Universal Robots PolyScope program: align_for_step.urp

Program align_for_step (installation=default directory=/programs createdIn=5.21.3 lastSavedIn=5.21.3 robotSerialNumber=20246801938)
Calibrated DH parameters: a=[-0.000071, -0.790281, -0.600694, 0.000061, -0.000039, 0]; d=[0.236272, 604.465945, 132.116513, -736.382239, 0.159268, 0.154005]; alpha=[1.570254, -0.000567, 0.000559, 1.571709, -1.56999, 0]; deltaTheta=[0, -0.409357, 7.293326, -0.600784, -0.000001, -0.000001]
InitVariablesNode
Robot Program (runOnlyOnce=false)
  'first move block is unnecessay and bad'
  SuppressedNode
    MoveJ speed 60 deg/s, acceleration 80 deg/s^2 (useActiveTCP=true optimoveEnabled=false optiMoveSpeed=0.3 optiMoveAcceleration=0.09) feature=Base
      'belowis oldhome'
      Waypoint Waypoint_1: TCP in base x=397.354 y=356.263 z=319.809 mm, rx=2.3163 ry=2.0576 rz=0.0741 rad; joints [-198.308, -118.162, 133.452, -12.561, -11.517, -6.326] deg; TCP offset x=-9.5 y=-328 z=105.73 mm, rx=1.2092 ry=-1.2092 rz=1.2092 rad
      SuppressedNode
        Waypoint Waypoint_2: TCP in base x=102.072 y=804.129 z=-21.158 mm, rx=-1.0098 ry=-2.9661 rz=0.0347 rad; joints [-131.791, -72.228, 126.432, -52.794, -4.122, -0.058] deg
      SuppressedNode
        Waypoint Waypoint_3: TCP in base x=-481.576 y=738.776 z=-387.745 mm, rx=-0.0268 ry=3.1371 rz=-0.1325 rad; joints [-88.373, -42.244, 121.849, -79.055, 0.705, 4.289] deg
      Waypoint Waypoint_4: TCP in base x=-790.625 y=220.046 z=-730.503 mm, rx=-0.9425 ry=2.9648 rz=-0.1356 rad; joints [-49.775, -15.59, 117.776, -102.401, 4.996, 5.448] deg
      Waypoint Waypoint_5: TCP in base x=-802.158 y=237.168 z=-730.663 mm, rx=0.8868 ry=-2.4516 rz=0.2829 rad; joints [-61.24, 14.733, 101.407, -222.645, 33.575, 110.967] deg
      Waypoint Waypoint_6: TCP in base x=-687.678 y=589.975 z=-233.622 mm, rx=-0.3444 ry=-1.0001 rz=-2.0808 rad; joints [-61.24, 14.733, 101.407, -222.645, 33.575, -30.853] deg
      SuppressedNode
        Waypoint goalpt: TCP in base x=-796.965 y=229.005 z=-75.004 mm, rx=0 ry=0 rz=-2.526 rad; joints [-49.775, -15.59, 117.776, -102.401, 4.996, -179.788] deg
      Waypoint goalpt2: TCP in base x=-1080.054 y=352.633 z=-86.722 mm, rx=0.0341 ry=-0.0008 rz=-2.631 rad; joints [-41.761, 5.394, 77.547, 101.81, -19.08, -4.137] deg
      Waypoint dummythere: TCP in base x=-1288.589 y=229.005 z=-75.004 mm, rx=0 ry=0 rz=-2.526 rad; joints [-29.748, -12.575, 79.071, -66.58, 25.031, -179.927] deg
  'second one is good'
  SuppressedNode
    MoveJ speed 60 deg/s, acceleration 80 deg/s^2 (useActiveTCP=true optimoveEnabled=false optiMoveSpeed=0.3 optiMoveAcceleration=0.09) feature=Base
      Waypoint goalpt2: TCP in base x=-1080.054 y=352.633 z=-86.722 mm, rx=0.0341 ry=-0.0008 rz=-2.631 rad; joints [-41.761, 5.394, 77.547, 101.81, -19.08, -4.137] deg
  'above was for wrong weldpath'
  SuppressedNode
    Folder savepoints
      MoveJ speed 60 deg/s, acceleration 80 deg/s^2 (useActiveTCP=true optimoveEnabled=false optiMoveSpeed=0.3 optiMoveAcceleration=0.09) feature=Base
        Waypoint leftstart: TCP in base x=-1168.534 y=251.879 z=303.712 mm, rx=-1.4388 ry=-0.6695 rz=0.6003 rad; joints [-161.388, -128.913, -89.606, -145.038, 61.894, 92.57] deg
  SuppressedNode
    MoveJ speed 60 deg/s, acceleration 80 deg/s^2 (useActiveTCP=true optimoveEnabled=false optiMoveSpeed=0.3 optiMoveAcceleration=0.09) feature=Base
      'final point before pa1'
      Waypoint Waypoint_7: TCP in base x=-913.411 y=251.879 z=303.712 mm, rx=-1.2351 ry=-1.1043 rz=1.0523 rad; joints [-156.391, -105.358, -132.178, -128.187, 33.298, 95.672] deg
      'oldhome'
      Waypoint Waypoint_8: TCP in base x=397.354 y=356.263 z=319.809 mm, rx=2.3163 ry=2.0576 rz=0.0741 rad; joints [-198.308, -118.162, 133.452, -12.561, -11.517, -6.326] deg
  MoveJ speed 60 deg/s, acceleration 80 deg/s^2 (useActiveTCP=true optimoveEnabled=false optiMoveSpeed=0.3 optiMoveAcceleration=0.09) feature=Base
    'from oldhome, actual path'
    SuppressedNode
      Waypoint Waypoint_9: TCP in base x=683.137 y=304.628 z=775.294 mm, rx=1.9572 ry=1.7212 rz=0.4516 rad; joints [-193.46, -116.682, 102.732, -25.933, -6.334, 5.47] deg
    SuppressedNode
      Waypoint Waypoint_10: TCP in base x=-197.847 y=491.143 z=1723.576 mm, rx=-0.0125 ry=0.2444 rz=1.7982 rad; joints [-175.692, -50.406, -94.795, -74.947, 12.663, 48.707] deg
    Waypoint Waypoint_11: TCP in base x=-557.589 y=419.56 z=1207.727 mm, rx=-0.5026 ry=-0.0558 rz=1.8139 rad; joints [-165.719, -50.766, -121.227, -102.266, 18.039, 76.633] deg
    SuppressedNode
      Waypoint Waypoint_12: TCP in base x=-793.876 y=251.879 z=303.712 mm, rx=-1.2351 ry=-1.1043 rz=1.0523 rad; joints [-150.736, -98.884, -141.754, -124.357, 38.932, 94.772] deg
  MoveL speed 250 mm/s, acceleration 50 mm/s^2 (useActiveTCP=true optimoveEnabled=false optiMoveSpeed=0.3 optiMoveAcceleration=0.09) feature=Base
    Waypoint Waypoint_12: TCP in base x=-793.876 y=251.879 z=303.712 mm, rx=-1.2351 ry=-1.1043 rz=1.0523 rad; joints [-150.736, -98.884, -141.754, -124.357, 38.932, 94.772] deg
